FUNCTION_BLOCK UnitTestWithOneMatchingAndOneNonMatchingName EXTENDS FB_TestSuite

HasMatchingName();
NameDoesntMatch();

METHOD HasMatchingName
TEST('HasMatchingName');

AssertTrue(Condition:=TRUE, Message:='Blabla');

TEST_FINISHED();
END_METHOD

METHOD NameDoesntMatch
VAR_INPUT
END_VAR
TEST('TheNameCertainlyDoesntMatch');

AssertTrue(Condition:=TRUE, Message:='Blabla');

TEST_FINISHED();
END_METHOD

END_FUNCTION_BLOCK

(* stored: Version 1.1.0.1, ProductVersion 3.1.4024.12
   POU UnitTestWithOneMatchingAndOneNonMatchingName: Id {66a0debc-b9cd-4b27-a180-e0a3969004d0}, SpecialFunc None
   Method HasMatchingName: Id {e8f9cfce-1f1c-44f4-93fb-68e8399c5ca1}
   Method NameDoesntMatch: Id {bb46751f-6e32-418e-b8a1-e16c822e22b2} *)
